ABB RobotStudio station: InjectorSetUp.rsstnx

Station InjectorSetUp (saved by RobotStudio 24.4.11080.0)
Controller IRB4600_60_205_2
  mechanical unit ROB_1: IRB4600_60_205_C_01, 6 joints, base frame (0, 0, 0) mm
Layout (positions relative to the parent item):
  - 1. AttacherBlackL [smart component, from Components\Attacher.rslib] at (-1000, 0, 0) mm
      properties: Parent=MoldGripper; Flange=0; Child=1. BlackL; Mount=false; Offset=[0 0 0]; Orientation=[0 0 0]
  - 1. TakeSensorBlackL [smart component, from Components\LineSensor.rslib] at (-1000, 295, -84.5) mm
      properties: Start=[0.95 1.25 1.44146]; End=[1.05 1.25 1.44146]; Length=0.1; Radius=0; Tag=(none); SensedPart=(none); SensedPoint=[0 0 0]
    - _sensorPart_ [part], size 100 x 0 x 0 mm
  - 1. PosBlackL [smart component, from Components\Positioner.rslib] at (-1000, 300, 0) mm
      properties: Object=1. BlackL; Position=[-0.25 1.55 1.5]; Orientation=[0 0 0]; Reference=Global; ReferenceObject=(none)
  - 1. DetacherBlackL [smart component, from Components\Detacher.rslib] at (-1000, 300, 0) mm
      properties: Child=1. BlackL; KeepPosition=true
  - 0. DropSensorBaseL [smart component, from Components\LineSensor.rslib] at (-1500, -37.49, 0) mm
      properties: Start=[3.2 0.43748 1.53501]; End=[2.7 0.43748 1.53501]; Length=0.5; Radius=0; Tag=(none); SensedPart=(none); SensedPoint=[0 0 0]
    - _sensorPart_ [part], size 500 x 0 x 0 mm
  - 1. PosBlackR [smart component, from Components\Positioner.rslib] at (-1000, -300, 0) mm
      properties: Object=1. BlackR; Position=[0.25 -1.55 1.5]; Orientation=[0 0 3.14159265358979]; Reference=Global; ReferenceObject=(none)
  - 1. AttacherBlackR [smart component, from Components\Attacher.rslib] at (-1000, -100, 0) mm
      properties: Parent=MoldGripper; Flange=0; Child=1. BlackR; Mount=false; Offset=[0 0 0]; Orientation=[0 0 0]
  - 1. TakeSensorBlackR [smart component, from Components\LineSensor.rslib] at (-1150, -300, -91.46) mm
      properties: Start=[1.1 -1.245 1.44842]; End=[1.2 -1.245 1.44842]; Length=0.1; Radius=0; Tag=(none); SensedPart=(none); SensedPoint=[0 0 0]
    - _sensorPart_ [part], size 100 x 0 x 0 mm
  - 0. TakeSensorBaseR [smart component, from Components\LineSensor.rslib] at (-1500, -800, -91.46) mm
      properties: Start=[3 0.605 1.54842]; End=[2.9 0.605 1.54842]; Length=0.0999999999999996; Radius=0; Tag=(none); SensedPart=(none); SensedPoint=[0 0 0]
    - _sensorPart_ [part], size 100 x 0 x 0 mm
  - 1. DetacherBlackR [smart component, from Components\Detacher.rslib] at (-1000, -300, 0) mm
      properties: Child=1. BlackR; KeepPosition=true
  - 2. AttacherRedL [smart component, from Components\Attacher.rslib] at (-1420, 300, 0) mm
      properties: Parent=MoldGripper; Flange=0; Child=2. RedL; Mount=false; Offset=[0 0 0]; Orientation=[0 0 0]
  - 2. TakeSensorRedL [smart component, from Components\LineSensor.rslib] at (-1150, 300, -91.46) mm
      properties: Start=[1.1 1.245 0.94842]; End=[1.2 1.245 0.94842]; Length=0.1; Radius=0; Tag=(none); SensedPart=(none); SensedPoint=[0 0 0]
    - _sensorPart_ [part], size 100 x 0 x 0 mm
  - 2. PosRedL [smart component, from Components\Positioner.rslib] at (-1420, 100, 0) mm
      properties: Object=2. RedL; Position=[-0.25 1.55 1]; Orientation=[0 0 0]; Reference=Global; ReferenceObject=(none)
  - 2. DetacherRedL [smart component, from Components\Detacher.rslib] at (-1420, 300, 0) mm
      properties: Child=2. RedL; KeepPosition=true
  - 2. PosRedR [smart component, from Components\Positioner.rslib] at (-1420, -300, 0) mm
      properties: Object=2. RedR; Position=[0.25 -1.55 1]; Orientation=[0 0 3.14159265358979]; Reference=Global; ReferenceObject=(none)
  - 2. AttacherRedR [smart component, from Components\Attacher.rslib] at (-1420, -300, 0) mm
      properties: Parent=MoldGripper; Flange=0; Child=2. RedR; Mount=false; Offset=[0 0 0]; Orientation=[0 0 0]
  - 2. TakeSensorRedR [smart component, from Components\LineSensor.rslib] at (-1570, -300, -91.46) mm
      properties: Start=[1.52 -1.245 0.94842]; End=[1.62 -1.245 0.94842]; Length=0.1; Radius=0; Tag=(none); SensedPart=(none); SensedPoint=[0 0 0]
    - _sensorPart_ [part], size 100 x 0 x 0 mm
  - 2. DetacherRedR [smart component, from Components\Detacher.rslib] at (-1420, -300, 0) mm
      properties: Child=2. RedR; KeepPosition=true
  - 3. AttacherBlueL [smart component, from Components\Attacher.rslib] at (-1840, 300, 0) mm
      properties: Parent=MoldGripper; Flange=0; Child=3. BlueL; Mount=false; Offset=[0 0 0]; Orientation=[0 0 0]
  - 3. TakeSensorBlueL [smart component, from Components\LineSensor.rslib] at (-1150, 300, -91.46) mm
      properties: Start=[1.1 1.245 0.44842]; End=[1.2 1.245 0.44842]; Length=0.1; Radius=0; Tag=(none); SensedPart=(none); SensedPoint=[0 0 0]
    - _sensorPart_ [part], size 100 x 0 x 0 mm
  - 3. PosBlueL [smart component, from Components\Positioner.rslib] at (-1840, 300, 0) mm
      properties: Object=3. BlueL; Position=[-0.25 1.55 0.5]; Orientation=[0 0 0]; Reference=Global; ReferenceObject=(none)
  - 3. DetacherBlueL [smart component, from Components\Detacher.rslib] at (-1840, 300, 0) mm
      properties: Child=3. BlueL; KeepPosition=true
  - 3. PosBlueR [smart component, from Components\Positioner.rslib] at (-1840, -300, 0) mm
      properties: Object=3. BlueR; Position=[0.25 -1.55 0.5]; Orientation=[0 0 3.14159265358979]; Reference=Global; ReferenceObject=(none)
  - 3. AttacherBlueR [smart component, from Components\Attacher.rslib] at (-1840, -300, 0) mm
      properties: Parent=MoldGripper; Flange=0; Child=3. BlueR; Mount=false; Offset=[0 0 0]; Orientation=[0 0 0]
  - 3. TakeSensorBlueR [smart component, from Components\LineSensor.rslib] at (-1990, -300, -91.46) mm
      properties: Start=[1.94 -1.245 0.44842]; End=[2.04 -1.245 0.44842]; Length=0.1; Radius=0; Tag=(none); SensedPart=(none); SensedPoint=[0 0 0]
    - _sensorPart_ [part], size 100 x 0 x 0 mm
  - 3. DetacherBlueR [smart component, from Components\Detacher.rslib] at (-1840, -300, 0) mm
      properties: Child=3. BlueR; KeepPosition=true
  - InjectionMachine [part] at (900, 1700, 0) mm, size 1314.8 x 3413.3 x 1819.5 mm
  - ClosePressFunction [smart component, from Components\JointMover.rslib] at (-1000, 0, 0) mm
      properties: Mechanism=Press; Relative=false; Duration=0.5; J1=0.4
  - OpenPressFunction [smart component, from Components\JointMover.rslib] at (-1000, 0, 0) mm
      properties: Mechanism=Press; Relative=false; Duration=0.5; J1=0
  - 0. DropSensorBaseR [smart component, from Components\LineSensor.rslib] at (-1500, -800, 50) mm
      properties: Start=[3.2 0.40001 1.48501]; End=[2.7 0.40001 1.48501]; Length=0.5; Radius=0; Tag=(none); SensedPart=2. RedR; SensedPoint=[1.20000036621094 -0.399989990234375 1.53501000976562]
    - _sensorPart_ [part], size 500 x 0 x 0 mm
  - 0. AttacherBaseRBlackR [smart component, from Components\Attacher.rslib] at (-1300, 0, 0) mm
      properties: Parent=Press; Flange=0; Child=1. BlackR; Mount=false; Offset=[0 0 0]; Orientation=[0 0 0]
  - 0. AttacherBaseRBlueR [smart component, from Components\Attacher.rslib] at (-1300, 0, 0) mm
      properties: Parent=Press; Flange=0; Child=3. BlueR; Mount=false; Offset=[0 0 0]; Orientation=[0 0 0]
  - 0. AttacherBaseRedR [smart component, from Components\Attacher.rslib] at (-1300, 0, 0) mm
      properties: Parent=Press; Flange=0; Child=2. RedR; Mount=false; Offset=[0 0 0]; Orientation=[0 0 0]
  - BlackRight [smart component, from Components\LogicGate.rslib]
      properties: Operator=AND; Delay=0
  - RedRight [smart component, from Components\LogicGate.rslib]
      properties: Operator=AND; Delay=0
  - BlueRight [smart component, from Components\LogicGate.rslib]
      properties: Operator=AND; Delay=0
  - 1. VolumeBlackR [smart component, from Components\VolumeSensor.rslib] at (-1020, -280, -20) mm
      properties: CornerPoint=[0.75 -1.25 1.1]; Orientation=[0 0 -1.5707963267949]; Length=0.24; Width=0.54; Height=0.44; Tag=(none); PartialHit=false; SensedPart=1. BlackR
    - _sensorPart_ [part], size 540 x 240 x 440 mm
  - BlackRight [smart component, from Components\LogicGate.rslib]
      properties: Operator=NOT; Delay=0
  - 2. VolumeRedR [smart component, from Components\VolumeSensor.rslib] at (-1020, -280, -520) mm
      properties: CornerPoint=[0.75 -1.25 1.1]; Orientation=[0 0 -1.5707963267949]; Length=0.24; Width=0.54; Height=0.44; Tag=(none); PartialHit=false; SensedPart=(none)
    - _sensorPart_ [part], size 540 x 240 x 440 mm
  - 3. VolumeBlueR [smart component, from Components\VolumeSensor.rslib] at (-1020, -280, -1020) mm
      properties: CornerPoint=[0.75 -1.25 1.1]; Orientation=[0 0 -1.5707963267949]; Length=0.24; Width=0.54; Height=0.44; Tag=(none); PartialHit=false; SensedPart=3. BlueR
    - _sensorPart_ [part], size 540 x 240 x 440 mm
  - RedRight [smart component, from Components\LogicGate.rslib]
      properties: Operator=NOT; Delay=0
  - BlueRight [smart component, from Components\LogicGate.rslib]
      properties: Operator=NOT; Delay=0
  - 0. VolumeBaseR [smart component, from Components\VolumeSensor.rslib] at (-1800, 840, 0) mm
      properties: CornerPoint=[2.99 -1.03 1.19]; Orientation=[0 0 -1.5707963267949]; Length=0.215; Width=0.515; Height=0.415; Tag=(none); PartialHit=false; SensedPart=2. RedR
    - _sensorPart_ [part], size 515 x 215 x 415 mm
  - 0. VolumeBaseL [smart component, from Components\VolumeSensor.rslib] at (-1800, 1000, 0) mm
      properties: CornerPoint=[3.51 -0.81 1.19]; Orientation=[0 0 1.5707963267949]; Length=0.215; Width=0.515; Height=0.415; Tag=(none); PartialHit=false; SensedPart=(none)
    - _sensorPart_ [part], size 515 x 215 x 415 mm
  - TakeRight [smart component, from Components\LogicGate.rslib]
      properties: Operator=AND; Delay=0
  - TakeRight [smart component, from Components\LogicGate.rslib]
      properties: Operator=NOT; Delay=0
  - BaseBlackRight [smart component, from Components\LogicGate.rslib]
      properties: Operator=AND; Delay=0
  - 0. PosBaseBlackR [smart component, from Components\Positioner.rslib] at (-1300, 0, 0) mm
      properties: Object=1. BlackR; Position=[1.7 -0.2 1.6]; Orientation=[0 0 -3.14159265358979]; Reference=Global; ReferenceObject=(none)
  - 0. PosBaseBlackL [smart component, from Components\Positioner.rslib] at (-1300, 0, 0) mm
      properties: Object=1. BlackL; Position=[1.2 0.2 1.6]; Orientation=[0 0 0]; Reference=Global; ReferenceObject=(none)
  - TakeLeft [smart component, from Components\LogicGate.rslib]
      properties: Operator=AND; Delay=0
  - BaseBlackLeft [smart component, from Components\LogicGate.rslib]
      properties: Operator=AND; Delay=0
  - 0. TakeSensorBaseL [smart component, from Components\LineSensor.rslib] at (-1500, -420, -91.46) mm
      properties: Start=[3 0.615 1.54842]; End=[2.9 0.615 1.54842]; Length=0.1; Radius=0; Tag=(none); SensedPart=(none); SensedPoint=[0 0 0]
    - _sensorPart_ [part], size 100 x 0 x 0 mm
  - 1. VolumeBlackL [smart component, from Components\VolumeSensor.rslib] at (-880, 280, -20) mm
      properties: CornerPoint=[1.15 1.25 1.1]; Orientation=[0 0 1.5707963267949]; Length=0.24; Width=0.54; Height=0.44; Tag=(none); PartialHit=false; SensedPart=1. BlackL
    - _sensorPart_ [part], size 540 x 240 x 440 mm
  - 2. VolumeRedL [smart component, from Components\VolumeSensor.rslib] at (-880, 280, -520) mm
      properties: CornerPoint=[1.15 1.25 1.1]; Orientation=[0 0 1.5707963267949]; Length=0.24; Width=0.54; Height=0.44; Tag=(none); PartialHit=false; SensedPart=(none)
    - _sensorPart_ [part], size 540 x 240 x 440 mm
  - 3. VolumeBlueL [smart component, from Components\VolumeSensor.rslib] at (-880, 280, -1020) mm
      properties: CornerPoint=[1.15 1.25 1.1]; Orientation=[0 0 1.5707963267949]; Length=0.24; Width=0.54; Height=0.44; Tag=(none); PartialHit=false; SensedPart=3. BlueL
    - _sensorPart_ [part], size 540 x 240 x 440 mm
  - BlackLeft [smart component, from Components\LogicGate.rslib]
      properties: Operator=NOT; Delay=0
  - RedLeft [smart component, from Components\LogicGate.rslib]
      properties: Operator=NOT; Delay=0
  - BlueLeft [smart component, from Components\LogicGate.rslib]
      properties: Operator=NOT; Delay=0
  - 1. DropSensorBlackL [smart component, from Components\LineSensor.rslib] at (-1000, -221.01, 0) mm
      properties: Start=[0.75 1.971 1.436]; End=[0.85 1.971 1.436]; Length=0.1; Radius=0; Tag=(none); SensedPart=1. BlackL; SensedPoint=[-0.249999877929688 1.74998999023437 1.436]
    - _sensorPart_ [part], size 100 x 0 x 0 mm
  - 1. DropSensorBlackR [smart component, from Components\LineSensor.rslib] at (-1200, -820.98, 0) mm, rotated rx 0 ry 0.01 rz 0 deg
      properties: Start=[1.44974952316885 -0.92901 1.43525305088395]; End=[0.949749530784283 -0.92901 1.4351657844218]; Length=0.5; Radius=0; Tag=(none); SensedPart=1. BlackR; SensedPoint=[0.25 -1.74998999023437 1.435]
    - _sensorPart_ [part], size 500 x 0 x 0.1 mm
  - 2. DropSensorRedR [smart component, from Components\LineSensor.rslib] at (-1200, -820.98, -500) mm, rotated rx 0 ry 0.01 rz 0 deg
      properties: Start=[1.44974952316885 -0.92901 1.43525305088395]; End=[0.949749530784283 -0.92901 1.4351657844218]; Length=0.5; Radius=0; Tag=(none); SensedPart=(none); SensedPoint=[0 0 0]
    - _sensorPart_ [part], size 500 x 0 x 0.1 mm
  - 2. DropSensorRedL [smart component, from Components\LineSensor.rslib] at (-1000, -221.01, -500) mm
      properties: Start=[0.75 1.971 1.435]; End=[1.25 1.971 1.435]; Length=0.5; Radius=0; Tag=(none); SensedPart=(none); SensedPoint=[0 0 0]
    - _sensorPart_ [part], size 500 x 0 x 0 mm
  - 3. DropSensorBlueR [smart component, from Components\LineSensor.rslib] at (-1200, -820.98, -1000) mm, rotated rx 0 ry 0.01 rz 0 deg
      properties: Start=[1.44974952316885 -0.92901 1.43525305088395]; End=[0.949749530784283 -0.92901 1.4351657844218]; Length=0.5; Radius=0; Tag=(none); SensedPart=3. BlueR; SensedPoint=[0.25 -1.74998999023437 0.435]
    - _sensorPart_ [part], size 500 x 0 x 0.1 mm
  - 3. DropSensorBlueL [smart component, from Components\LineSensor.rslib] at (-1000, -221.01, -1000) mm
      properties: Start=[0.75 1.971 1.435]; End=[1.25 1.971 1.435]; Length=0.5; Radius=0; Tag=(none); SensedPart=3. BlueL; SensedPoint=[0.249999969482422 1.74998999023437 0.435]
    - _sensorPart_ [part], size 500 x 0 x 0 mm
  - CloseSecurityTimer [smart component, from Components\Timer.rslib] at (-1000, 0, 0) mm
      properties: StartTime=1; Interval=0; Repeat=false; CurrentTime=0
  - InjectionCycleTimer [smart component, from Components\Timer.rslib]
      properties: StartTime=15.5; Interval=0; Repeat=false; CurrentTime=0
  - LogicSRLatch [smart component, from Components\LogicSRLatch.rslib]
  - BaseRedRight [smart component, from Components\LogicGate.rslib]
      properties: Operator=AND; Delay=0
  - BaseRedLeft [smart component, from Components\LogicGate.rslib]
      properties: Operator=AND; Delay=0
  - BaseBlueRight [smart component, from Components\LogicGate.rslib]
      properties: Operator=AND; Delay=0
  - BaseBlueLeft [smart component, from Components\LogicGate.rslib]
      properties: Operator=AND; Delay=0
  - ResetTimerAux [smart component, from Components\Timer.rslib] at (-600, 0, 0) mm
      properties: StartTime=0.1; Interval=0; Repeat=false; CurrentTime=192.816
  - IRB4600_60_205_C_01 [mechanism, from %ABB.RobotStudio.Models.IRB4600%\IRB4600_60_205_C_G_01.rslib] at (0, 0, 0) mm; joint values [1.5708, 0.4406, 0.2713, 0, -0.7118, 0] (rad or m)
  - OutMold1 [part] at (1510.58, -210, 320) mm, size 400 x 400 x 50 mm
  - FirstConveyor [part] at (1000, 190, 200) mm, size 2000 x 500 x 900 mm
  - MovementOutMold1 [smart component, from Components\MoveAlongCurve.rslib]
      properties: Object=OutMold1; WirePart=WayOutMold1; Speed=0.5; KeepOrientation=false; StartDistance=0; ResetPosition=true; StartPosition=[[1 0 0 0] [0 1 0 0] [0 0 1 0] [1.74 -0.21 0.32 1]]
  - MovementOutMold2 [smart component, from Components\MoveAlongCurve.rslib]
      properties: Object=OutMold2; WirePart=WayOutMold2; Speed=0.5; KeepOrientation=false; StartDistance=0; ResetPosition=false; StartPosition=[[1 0 0 0] [0 1 0 0] [0 0 1 0] [0 0 0 1]]
  - WayOutMold1 [part] at (-800, 0, 0) mm, size 240.6 x 0 x 0 mm
  - HideOutMold1 [smart component, from Components\Hide.rslib]
      properties: Object=OutMold1
  - HideOutMold2 [smart component, from Components\Hide.rslib]
      properties: Object=OutMold2
  - OutMold2 [part] at (2300.58, -211, 545) mm, rotated rx 0 ry -30 rz 0 deg, size 400 x 400 x 50 mm
  - ShowOutMold1 [smart component, from Components\Show.rslib] at (-600, 0, 0) mm
      properties: Object=OutMold1
  - ShowOutMold2 [smart component, from Components\Show.rslib] at (-600, 0, 0) mm
      properties: Object=OutMold2
  - WayOutMold2 [part] at (-600, 0, 0) mm, size 958.1 x 0 x 555.7 mm
  - PositionerOutMold1 [smart component, from Components\Positioner.rslib] at (-600, 0, 0) mm
      properties: Object=OutMold1; Position=[1.510578 -0.21 0.32]; Orientation=[0 0 0]; Reference=Global; ReferenceObject=(none)
  - PositionerOutMold2 [smart component, from Components\Positioner.rslib] at (-600, 0, 0) mm
      properties: Object=OutMold2; Position=[2.300578 -0.211 0.545]; Orientation=[0 -0.523598775598299 0]; Reference=Global; ReferenceObject=(none)
  - BlueColorOutMold1 [smart component, from Components\Highlighter.rslib]
      properties: Object=OutMold1; Color=[0 150 255]; Opacity=255
  - BlueColorOutMold2 [smart component, from Components\Highlighter.rslib]
      properties: Object=OutMold2; Color=[0 150 255]; Opacity=255
  - RedColorOutMold1 [smart component, from Components\Highlighter.rslib] at (-600, 0, 0) mm
      properties: Object=OutMold1; Color=[255 0 0]; Opacity=255
  - RedColorOutMold2 [smart component, from Components\Highlighter.rslib] at (-600, 0, 0) mm
      properties: Object=OutMold2; Color=[255 0 0]; Opacity=255
  - RedColorCount [smart component, from Components\Comparer.rslib] at (-600, 0, 0) mm
      properties: ValueA=2; Operator===; ValueB=1
  - CoreColorCounter [smart component, from Components\Counter.rslib]
      properties: Count=2
  - BlueColorCount [smart component, from Components\Comparer.rslib]
      properties: ValueA=2; Operator===; ValueB=2
  - ResetCoreCounter [smart component, from Components\Comparer.rslib] at (-600, 0, 0) mm
      properties: ValueA=2; Operator===; ValueB=3
  - OutMold1Sensor [smart component, from Components\LineSensor.rslib] at (-600, 0, 0) mm
      properties: Start=[1.910578 0.19 0.38]; End=[1.910578 -0.21 0.38]; Length=0.4; Radius=0; Tag=(none); SensedPart=(none); SensedPoint=[0 0 0]
    - _sensorPart_ [part], size 0 x 400 x 0 mm
  - RealOut [part] at (1610.58, -40, 1550) mm, rotated rx -90 ry 0 rz 0 deg, size 400 x 400 x 50 mm
  - MovementRealOutMold [smart component, from Components\LinearMover2.rslib]
      properties: Object=RealOut; Direction=[0 0 -0.001]; Distance=0.8; Duration=0.404; Reference=Global; ReferenceObject=(none)
  - PositionerRealOut [smart component, from Components\Positioner.rslib] at (-600, 0, 0) mm
      properties: Object=RealOut; Position=[1.610578 -0.04 1.55]; Orientation=[-1.5707963267949 0 0]; Reference=Global; ReferenceObject=(none)
  - ShowRealOutMold [smart component, from Components\Show.rslib] at (-600, 0, 0) mm
      properties: Object=RealOut
  - HideRealOut [smart component, from Components\Hide.rslib]
      properties: Object=RealOut
  - OpenPressAuxFunction [smart component, from Components\JointMover.rslib] at (-1000, 0, 0) mm
      properties: Mechanism=Press; Relative=false; Duration=0.5; J1=0
  - RedColorRealMold [smart component, from Components\Highlighter.rslib] at (-600, 0, 0) mm
      properties: Object=RealOut; Color=[255 0 0]; Opacity=255
  - BlueColorRealMold [smart component, from Components\Highlighter.rslib] at (-600, 0, 0) mm
      properties: Object=RealOut; Color=[0 150 255]; Opacity=255
  - IRC5_Single-Cabinet [part, from %ABB.RobotStudio.Models.IRC5%\IRC5_Single-Cabinet.rslib] at (-3450, 450, 100) mm, rotated rx 90 ry 0 rz -90 deg
  - FlexPendant [part, from %ABB.RobotStudio.Models.IRC5%\FlexPendant.rslib] at (-3350, 630, 990) mm, rotated rx -27.17 ry 5.43 rz -119.59 deg
  - EnablingSwitch [part] at (-3520, 650, 920) mm, rotated rx 0 ry 0 rz 180 deg, size 62.9 x 279 x 47.8 mm
  - MoldGripper [mechanism] at (0, 1535, 814.49) mm, rotated rx 0 ry 90 rz 90 deg
      TCP MoldGripper at (0, -85, -10.5) mm, rotated rx 0 ry -90 rz 90 deg
      links: EndEffector
  - 0. BaseMoldL [part] at (-300, 0, 4000) mm, size 500 x 200 x 400 mm
  - Press [mechanism] at (-300, 0, 0) mm; joint values [0] (rad or m)
      links: Link1, Link2
  - 3. BlueL [part] at (-250, 1550, 498.43) mm, size 500 x 200 x 400 mm
  - 2. RedL [part] at (-250, 1550, 1019.95) mm, size 500 x 200 x 400 mm
  - 1. BlackL [part] at (-250, 1550, 1500.71) mm, size 500 x 200 x 400 mm
  - 1. BlackR [part] at (250, -1550, 1500) mm, rotated rx 0 ry 0 rz 180 deg, size 500 x 200 x 400 mm
  - 2. RedR [part] at (1700, -200, 1599.37) mm, rotated rx 0 ry 0 rz -180 deg, size 500 x 200 x 400 mm
  - 3. BlueR [part] at (250, -1550, 500) mm, rotated rx 0 ry 0 rz 180 deg, size 500 x 200 x 400 mm
  - MoldStore [part] at (285, 1550, 0) mm, rotated rx 0 ry 0 rz 90 deg, size 300 x 610 x 1600 mm
  - MoldStore_2 [part] at (-285, -1550, 0) mm, rotated rx 0 ry 0 rz -90 deg, size 300 x 610 x 1600 mm
  - Fence_3 [graphiccomponentgroup]
    - Segment 1 [part], size 169.7 x 169.7 x 1400 mm
    - Segment 2 [part], size 316.7 x 1054.9 x 1400 mm
    - Segment 3 [part], size 169.7 x 1684.9 x 1400 mm
    - Segment 3 [part], size 169.7 x 1684.9 x 1400 mm
    - Segment 3 [part], size 169.7 x 1684.9 x 1400 mm
  - Fence_2 [graphiccomponentgroup]
    - Segment 1 [part], size 169.7 x 169.7 x 1400 mm
    - Segment 2 [part], size 1959.9 x 169.7 x 1400 mm
    - Segment 2 [part], size 1959.9 x 169.7 x 1400 mm
  - Fence [graphiccomponentgroup]
    - Segment 1 [part], size 169.7 x 169.7 x 1400 mm
    - Segment 2 [part], size 1959.9 x 169.7 x 1400 mm
    - Segment 2 [part], size 1959.9 x 169.7 x 1400 mm
  - Fence_6 [graphiccomponentgroup]
    - Segment 1 [part], size 169.7 x 169.7 x 2000 mm
    - Segment 2 [part], size 169.7 x 1134.9 x 2000 mm
    - Segment 2 [part], size 169.7 x 1134.9 x 2000 mm
  - Fence_4 [graphiccomponentgroup]
    - Segment 1 [part], size 169.7 x 169.7 x 2000 mm
    - Segment 2 [part], size 169.7 x 1134.9 x 2000 mm
    - Segment 2 [part], size 169.7 x 1134.9 x 2000 mm
  - Fence_5 [graphiccomponentgroup]
    - Segment 1 [part], size 169.7 x 169.7 x 1400 mm
    - Segment 2 [part], size 169.7 x 169.7 x 1400 mm
  - Pieza_3 [part], size 15 x 940 x 15 mm
  - Pieza_4 [part] at (0, 0, 500) mm, size 15 x 940 x 15 mm
  - Pieza_5 [part] at (0, 0, -500) mm, size 15 x 940 x 15 mm
  - ControlPanel [part] at (-3165, 1650, 600) mm, rotated rx 0 ry 0 rz -90 deg, size 600 x 300 x 800 mm
  - ModeSelecting1 [smart component, from Components\LogicMux.rslib]
  - ModeSelecting2 [smart component, from Components\LogicMux.rslib]
  - ModeCounter [smart component, from Components\Counter.rslib]
      properties: Count=5
Attachment: MoldGripper is attached to IRB4600_60_205_C_01 / Link6
Attachment: 2. RedR is attached to Press / Link2
Attachment: 2. RedL is attached to MoldGripper / EndEffector
Station signals: DI Digital1, DI Digital2
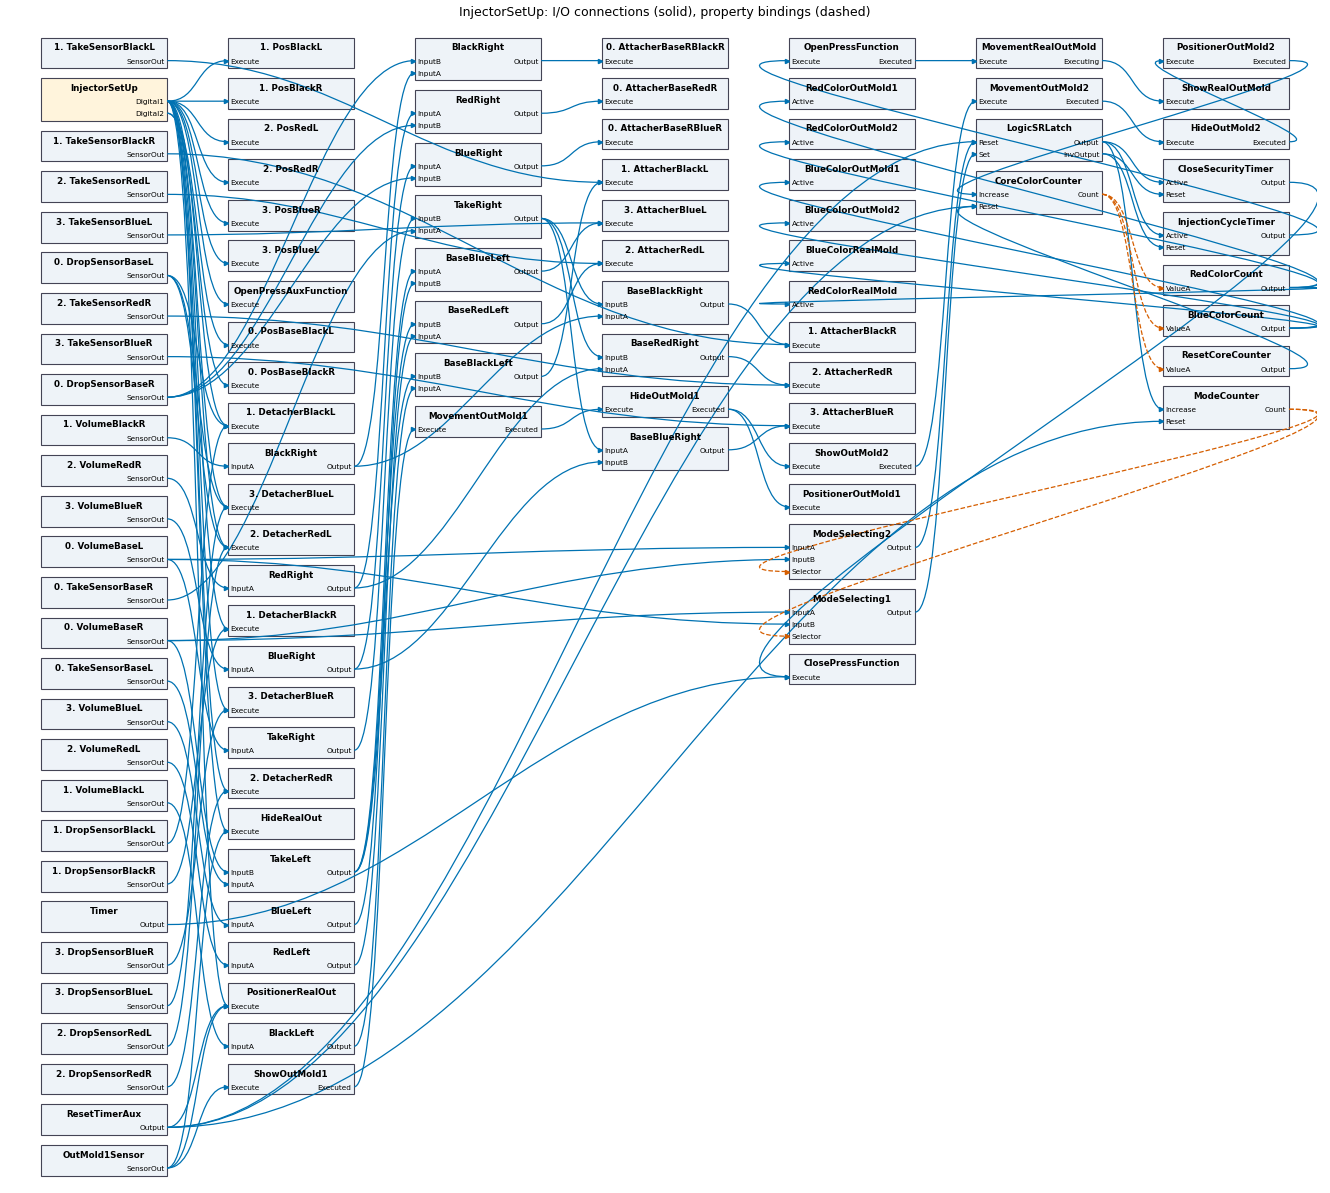
Station logic (signal -> signal, property => property):
  1. TakeSensorBlackL.SensorOut -> 1. AttacherBlackL.Execute
  InjectorSetUp.Digital1 -> 1. PosBlackL.Execute
  InjectorSetUp.Digital1 -> 1. DetacherBlackL.Execute
  InjectorSetUp.Digital1 -> 1. PosBlackR.Execute
  1. TakeSensorBlackR.SensorOut -> 1. AttacherBlackR.Execute
  InjectorSetUp.Digital1 -> 1. DetacherBlackR.Execute
  InjectorSetUp.Digital1 -> 2. DetacherRedL.Execute
  InjectorSetUp.Digital1 -> 3. DetacherBlueL.Execute
  InjectorSetUp.Digital1 -> 2. DetacherRedR.Execute
  InjectorSetUp.Digital1 -> 3. DetacherBlueR.Execute
  2. TakeSensorRedL.SensorOut -> 2. AttacherRedL.Execute
  3. TakeSensorBlueL.SensorOut -> 3. AttacherBlueL.Execute
  0. DropSensorBaseL.SensorOut -> 1. DetacherBlackL.Execute
  0. DropSensorBaseL.SensorOut -> 2. DetacherRedL.Execute
  0. DropSensorBaseL.SensorOut -> 3. DetacherBlueL.Execute
  2. TakeSensorRedR.SensorOut -> 2. AttacherRedR.Execute
  3. TakeSensorBlueR.SensorOut -> 3. AttacherBlueR.Execute
  InjectorSetUp.Digital1 -> 2. PosRedL.Execute
  InjectorSetUp.Digital1 -> 2. PosRedR.Execute
  InjectorSetUp.Digital1 -> 3. PosBlueR.Execute
  InjectorSetUp.Digital1 -> 3. PosBlueL.Execute
  0. DropSensorBaseR.SensorOut -> BlackRight.InputB
  1. VolumeBlackR.SensorOut -> BlackRight.InputA
  BlackRight.Output -> BlackRight.InputA
  BlackRight.Output -> 0. AttacherBaseRBlackR.Execute
  2. VolumeRedR.SensorOut -> RedRight.InputA
  RedRight.Output -> RedRight.InputA
  RedRight.Output -> 0. AttacherBaseRedR.Execute
  3. VolumeBlueR.SensorOut -> BlueRight.InputA
  BlueRight.Output -> BlueRight.InputA
  0. DropSensorBaseR.SensorOut -> BlueRight.InputB
  0. DropSensorBaseR.SensorOut -> RedRight.InputB
  BlueRight.Output -> 0. AttacherBaseRBlueR.Execute
  0. VolumeBaseL.SensorOut -> TakeRight.InputA
  TakeRight.Output -> TakeRight.InputB
  0. TakeSensorBaseR.SensorOut -> TakeRight.InputA
  TakeRight.Output -> BaseBlackRight.InputB
  BaseBlackRight.Output -> 1. AttacherBlackR.Execute
  InjectorSetUp.Digital2 -> 0. PosBaseBlackL.Execute
  InjectorSetUp.Digital2 -> 0. PosBaseBlackR.Execute
  0. VolumeBaseR.SensorOut -> TakeLeft.InputB
  0. TakeSensorBaseL.SensorOut -> TakeLeft.InputA
  TakeLeft.Output -> BaseBlackLeft.InputB
  3. VolumeBlueL.SensorOut -> BlueLeft.InputA
  2. VolumeRedL.SensorOut -> RedLeft.InputA
  1. VolumeBlackL.SensorOut -> BlackLeft.InputA
  BlackLeft.Output -> BaseBlackLeft.InputA
  BaseBlackLeft.Output -> 1. AttacherBlackL.Execute
  BlackRight.Output -> BaseBlackRight.InputA
  1. DropSensorBlackL.SensorOut -> 1. DetacherBlackL.Execute
  1. DropSensorBlackR.SensorOut -> 1. DetacherBlackR.Execute
  Timer.Output -> ClosePressFunction.Execute
  CloseSecurityTimer.Output -> ClosePressFunction.Execute
  InjectionCycleTimer.Output -> OpenPressFunction.Execute
  LogicSRLatch.Output -> CloseSecurityTimer.Active
  LogicSRLatch.Output -> InjectionCycleTimer.Active
  LogicSRLatch.InvOutput -> InjectionCycleTimer.Reset
  LogicSRLatch.InvOutput -> CloseSecurityTimer.Reset
  3. DropSensorBlueR.SensorOut -> 3. DetacherBlueR.Execute
  3. DropSensorBlueL.SensorOut -> 3. DetacherBlueL.Execute
  2. DropSensorRedL.SensorOut -> 2. DetacherRedL.Execute
  2. DropSensorRedR.SensorOut -> 2. DetacherRedR.Execute
  TakeLeft.Output -> BaseRedLeft.InputB
  RedLeft.Output -> BaseRedLeft.InputA
  BaseRedLeft.Output -> 2. AttacherRedL.Execute
  TakeRight.Output -> BaseRedRight.InputB
  RedRight.Output -> BaseRedRight.InputA
  BaseRedRight.Output -> 2. AttacherRedR.Execute
  TakeLeft.Output -> BaseBlueLeft.InputA
  BlueLeft.Output -> BaseBlueLeft.InputB
  BaseBlueLeft.Output -> 3. AttacherBlueL.Execute
  TakeRight.Output -> BaseBlueRight.InputA
  BlueRight.Output -> BaseBlueRight.InputB
  BaseBlueRight.Output -> 3. AttacherBlueR.Execute
  ResetTimerAux.Output -> LogicSRLatch.Reset
  HideOutMold1.Executed -> ShowOutMold2.Execute
  ShowOutMold1.Executed -> MovementOutMold1.Execute
  ShowOutMold2.Executed -> MovementOutMold2.Execute
  MovementOutMold1.Executed -> HideOutMold1.Execute
  HideOutMold1.Executed -> PositionerOutMold1.Execute
  HideOutMold2.Executed -> PositionerOutMold2.Execute
  MovementOutMold2.Executed -> HideOutMold2.Execute
  PositionerOutMold2.Executed -> CoreColorCounter.Increase
  RedColorCount.Output -> RedColorOutMold1.Active
  RedColorCount.Output -> RedColorOutMold2.Active
  BlueColorCount.Output -> BlueColorOutMold1.Active
  BlueColorCount.Output -> BlueColorOutMold2.Active
  ResetTimerAux.Output -> CoreColorCounter.Reset
  ResetCoreCounter.Output -> CoreColorCounter.Reset
  OutMold1Sensor.SensorOut -> PositionerRealOut.Execute
  OutMold1Sensor.SensorOut -> ShowOutMold1.Execute
  ResetTimerAux.Output -> PositionerRealOut.Execute
  OpenPressFunction.Executed -> MovementRealOutMold.Execute
  InjectorSetUp.Digital1 -> PositionerRealOut.Execute
  OutMold1Sensor.SensorOut -> HideRealOut.Execute
  MovementRealOutMold.Executing -> ShowRealOutMold.Execute
  InjectorSetUp.Digital1 -> HideRealOut.Execute
  InjectorSetUp.Digital1 -> OpenPressAuxFunction.Execute
  BlueColorCount.Output -> BlueColorRealMold.Active
  RedColorCount.Output -> RedColorRealMold.Active
  0. VolumeBaseL.SensorOut -> ModeSelecting2.InputA
  ModeSelecting2.Output -> LogicSRLatch.Reset
  0. VolumeBaseR.SensorOut -> ModeSelecting2.InputB
  0. VolumeBaseR.SensorOut -> ModeSelecting1.InputA
  ModeSelecting1.Output -> LogicSRLatch.Set
  0. VolumeBaseL.SensorOut -> ModeSelecting1.InputB
  LogicSRLatch.Output -> ModeCounter.Increase
  ResetTimerAux.Output -> ModeCounter.Reset
  CoreColorCounter.Count => RedColorCount.ValueA
  CoreColorCounter.Count => BlueColorCount.ValueA
  CoreColorCounter.Count => ResetCoreCounter.ValueA
  ModeCounter.Count => ModeSelecting2.Selector
  ModeCounter.Count => ModeSelecting1.Selector
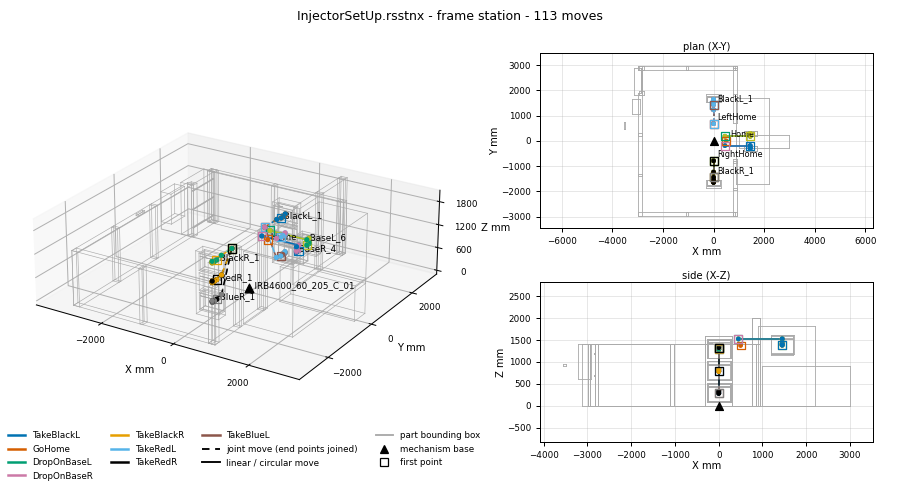
[picture p0: tool path of InjectorSetUp.rsstnx in frame station, 113 of 114 moves have a stored position in this frame; points joined in program order, loops and branches not executed]
Targets, tools, work objects and paths stored in the station, written as RAPID:
! task T_ROB1
MODULE Module1
  CONST jointtarget Rest:=[[0,-60,60,0,30,0],[9E+09,9E+09,9E+09,9E+09,9E+09,9E+09]];
  PROC GoRest()
    MoveAbsJ Rest,robotSpeed,z100,tool0\WObj:=wobj0;
  ENDPROC
  PROC TakeBlackL()
    MoveJ BlackL_1,robotSpeed,z100,MoldGripper\WObj:=LeftMoldStore;
    MoveL BlackL_2,robotSpeed,fine,MoldGripper\WObj:=LeftMoldStore;
    MoveL BlackL_3,robotSpeed,fine,MoldGripper\WObj:=LeftMoldStore;
    MoveL BlackL_4,robotSpeed,fine,MoldGripper\WObj:=LeftMoldStore;
    MoveL BlackL_5,robotSpeed,fine,MoldGripper\WObj:=LeftMoldStore;
    MoveL BlackL_6,robotSpeed,fine,MoldGripper\WObj:=LeftMoldStore;
    MoveJ LeftHome,robotSpeed,z100,MoldGripper\WObj:=LeftMoldStore;
  ENDPROC
  PROC GoHome()
    MoveJ Home,robotSpeed,z100,MoldGripper\WObj:=BaseMolds;
  ENDPROC
  PROC DropOnBaseL()
    MoveJ BaseL_7,robotSpeed,fine,MoldGripper\WObj:=BaseMolds;
    MoveL BaseL_6,robotSpeed,fine,MoldGripper\WObj:=BaseMolds;
    MoveL BaseL_5,robotSpeed,fine,MoldGripper\WObj:=BaseMolds;
    MoveL BaseL_4,robotSpeed,fine,MoldGripper\WObj:=BaseMolds;
    MoveL BaseL_3,robotSpeed,fine,MoldGripper\WObj:=BaseMolds;
    MoveL BaseL_2,robotSpeed,fine,MoldGripper\WObj:=BaseMolds;
    MoveL BaseL_1,robotSpeed,fine,MoldGripper\WObj:=BaseMolds;
  ENDPROC
  PROC DropOnBaseR()
    MoveJ BaseR_7,robotSpeed,fine,MoldGripper\WObj:=BaseMolds;
    MoveL BaseR_6,robotSpeed,fine,MoldGripper\WObj:=BaseMolds;
    MoveL BaseR_5,robotSpeed,fine,MoldGripper\WObj:=BaseMolds;
    MoveL BaseR_4,robotSpeed,fine,MoldGripper\WObj:=BaseMolds;
    MoveL BaseR_3,robotSpeed,fine,MoldGripper\WObj:=BaseMolds;
    MoveL BaseR_2,robotSpeed,fine,MoldGripper\WObj:=BaseMolds;
    MoveL BaseR_1,robotSpeed,fine,MoldGripper\WObj:=BaseMolds;
  ENDPROC
  PROC TakeBlackR()
    MoveJ BlackR_1,robotSpeed,z100,MoldGripper\WObj:=RightMoldStore;
    MoveL BlackR_2,robotSpeed,fine,MoldGripper\WObj:=RightMoldStore;
    MoveL BlackR_3,robotSpeed,fine,MoldGripper\WObj:=RightMoldStore;
    MoveL BlackR_4,robotSpeed,fine,MoldGripper\WObj:=RightMoldStore;
    MoveL BlackR_5,robotSpeed,fine,MoldGripper\WObj:=RightMoldStore;
    MoveL BlackR_6,robotSpeed,fine,MoldGripper\WObj:=RightMoldStore;
    MoveJ RightHome,robotSpeed,z100,MoldGripper\WObj:=RightMoldStore;
  ENDPROC
  PROC TakeRedL()
    MoveJ RedL_1,robotSpeed,z100,MoldGripper\WObj:=LeftMoldStore;
    MoveL RedL_2,robotSpeed,fine,MoldGripper\WObj:=LeftMoldStore;
    MoveL RedL_3,robotSpeed,fine,MoldGripper\WObj:=LeftMoldStore;
    MoveL RedL_4,robotSpeed,fine,MoldGripper\WObj:=LeftMoldStore;
    MoveL RedL_5,robotSpeed,fine,MoldGripper\WObj:=LeftMoldStore;
    MoveL RedL_6,robotSpeed,fine,MoldGripper\WObj:=LeftMoldStore;
    MoveJ LeftHome,robotSpeed,z100,MoldGripper\WObj:=LeftMoldStore;
  ENDPROC
  PROC TakeRedR()
    MoveJ RedR_1,robotSpeed,z100,MoldGripper\WObj:=RightMoldStore;
    MoveL RedR_2,robotSpeed,fine,MoldGripper\WObj:=RightMoldStore;
    MoveL RedR_3,robotSpeed,fine,MoldGripper\WObj:=RightMoldStore;
    MoveL RedR_4,robotSpeed,fine,MoldGripper\WObj:=RightMoldStore;
    MoveL RedR_5,robotSpeed,fine,MoldGripper\WObj:=RightMoldStore;
    MoveL RedR_6,robotSpeed,fine,MoldGripper\WObj:=RightMoldStore;
    MoveJ RightHome,robotSpeed,z100,MoldGripper\WObj:=RightMoldStore;
  ENDPROC
  PROC TakeBlueL()
    MoveJ BlueL_1,robotSpeed,z100,MoldGripper\WObj:=LeftMoldStore;
    MoveL BlueL_2,robotSpeed,fine,MoldGripper\WObj:=LeftMoldStore;
    MoveL BlueL_3,robotSpeed,fine,MoldGripper\WObj:=LeftMoldStore;
    MoveL BlueL_4,robotSpeed,fine,MoldGripper\WObj:=LeftMoldStore;
    MoveL BlueL_5,robotSpeed,fine,MoldGripper\WObj:=LeftMoldStore;
    MoveL BlueL_6,robotSpeed,fine,MoldGripper\WObj:=LeftMoldStore;
    MoveJ LeftHome,robotSpeed,z100,MoldGripper\WObj:=LeftMoldStore;
  ENDPROC
  PROC TakeBlueR()
    MoveJ BlueR_1,robotSpeed,z100,MoldGripper\WObj:=RightMoldStore;
    MoveL BlueR_2,robotSpeed,fine,MoldGripper\WObj:=RightMoldStore;
    MoveL BlueR_3,robotSpeed,fine,MoldGripper\WObj:=RightMoldStore;
    MoveL BlueR_4,robotSpeed,fine,MoldGripper\WObj:=RightMoldStore;
    MoveL BlueR_5,robotSpeed,fine,MoldGripper\WObj:=RightMoldStore;
    MoveL BlueR_6,robotSpeed,fine,MoldGripper\WObj:=RightMoldStore;
    MoveJ RightHome,robotSpeed,z100,MoldGripper\WObj:=RightMoldStore;
  ENDPROC
  PROC TakeFromBaseL()
    MoveJ BaseL_1,robotSpeed,z100,MoldGripper\WObj:=BaseMolds;
    MoveL BaseL_2,robotSpeed,fine,MoldGripper\WObj:=BaseMolds;
    MoveL BaseL_3,robotSpeed,fine,MoldGripper\WObj:=BaseMolds;
    MoveL BaseL_4,robotSpeed,fine,MoldGripper\WObj:=BaseMolds;
    MoveL BaseL_5,robotSpeed,fine,MoldGripper\WObj:=BaseMolds;
    MoveL BaseL_6,robotSpeed,fine,MoldGripper\WObj:=BaseMolds;
    MoveL BaseL_7,robotSpeed,fine,MoldGripper\WObj:=BaseMolds;
  ENDPROC
  PROC TakeFromBaseR()
    MoveJ BaseR_1,robotSpeed,z100,MoldGripper\WObj:=BaseMolds;
    MoveL BaseR_2,robotSpeed,fine,MoldGripper\WObj:=BaseMolds;
    MoveL BaseR_3,robotSpeed,fine,MoldGripper\WObj:=BaseMolds;
    MoveL BaseR_4,robotSpeed,fine,MoldGripper\WObj:=BaseMolds;
    MoveL BaseR_5,robotSpeed,fine,MoldGripper\WObj:=BaseMolds;
    MoveL BaseR_6,robotSpeed,fine,MoldGripper\WObj:=BaseMolds;
    MoveL BaseR_7,robotSpeed,fine,MoldGripper\WObj:=BaseMolds;
  ENDPROC
  PROC DropBlackL()
    MoveJ LeftHome,robotSpeed,z100,MoldGripper\WObj:=LeftMoldStore;
    MoveJ BlackL_6,robotSpeed,z100,MoldGripper\WObj:=LeftMoldStore;
    MoveL BlackL_5,robotSpeed,fine,MoldGripper\WObj:=LeftMoldStore;
    MoveL BlackL_4,robotSpeed,fine,MoldGripper\WObj:=LeftMoldStore;
    MoveL BlackL_3,robotSpeed,fine,MoldGripper\WObj:=LeftMoldStore;
    MoveL BlackL_2,robotSpeed,fine,MoldGripper\WObj:=LeftMoldStore;
    MoveJ BlackL_1,robotSpeed,z100,MoldGripper\WObj:=LeftMoldStore;
  ENDPROC
  PROC DropBlackR()
    MoveJ RightHome,robotSpeed,z100,MoldGripper\WObj:=RightMoldStore;
    MoveJ BlackR_6,robotSpeed,z100,MoldGripper\WObj:=RightMoldStore;
    MoveL BlackR_5,robotSpeed,fine,MoldGripper\WObj:=RightMoldStore;
    MoveL BlackR_4,robotSpeed,fine,MoldGripper\WObj:=RightMoldStore;
    MoveL BlackR_3,robotSpeed,fine,MoldGripper\WObj:=RightMoldStore;
    MoveL BlackR_2,robotSpeed,fine,MoldGripper\WObj:=RightMoldStore;
    MoveJ BlackR_1,robotSpeed,z100,MoldGripper\WObj:=RightMoldStore;
  ENDPROC
  PROC DropRedL()
    MoveJ LeftHome,robotSpeed,z100,MoldGripper\WObj:=LeftMoldStore;
    MoveJ RedL_6,robotSpeed,z100,MoldGripper\WObj:=LeftMoldStore;
    MoveL RedL_5,robotSpeed,fine,MoldGripper\WObj:=LeftMoldStore;
    MoveL RedL_4,robotSpeed,fine,MoldGripper\WObj:=LeftMoldStore;
    MoveL RedL_3,robotSpeed,fine,MoldGripper\WObj:=LeftMoldStore;
    MoveL RedL_2,robotSpeed,fine,MoldGripper\WObj:=LeftMoldStore;
    MoveJ RedL_1,robotSpeed,z100,MoldGripper\WObj:=LeftMoldStore;
  ENDPROC
  PROC DropRedR()
    MoveJ RightHome,v7000,z100,MoldGripper\WObj:=RightMoldStore;
    MoveJ RedR_6,robotSpeed,z100,MoldGripper\WObj:=RightMoldStore;
    MoveL RedR_5,robotSpeed,fine,MoldGripper\WObj:=RightMoldStore;
    MoveL RedR_4,robotSpeed,fine,MoldGripper\WObj:=RightMoldStore;
    MoveL RedR_3,robotSpeed,fine,MoldGripper\WObj:=RightMoldStore;
    MoveL RedR_2,robotSpeed,fine,MoldGripper\WObj:=RightMoldStore;
    MoveJ RedR_1,robotSpeed,z100,MoldGripper\WObj:=RightMoldStore;
  ENDPROC
  PROC DropBlueL()
    MoveJ LeftHome,robotSpeed,z100,MoldGripper\WObj:=LeftMoldStore;
    MoveJ BlueL_6,robotSpeed,z100,MoldGripper\WObj:=LeftMoldStore;
    MoveL BlueL_5,robotSpeed,fine,MoldGripper\WObj:=LeftMoldStore;
    MoveL BlueL_4,robotSpeed,fine,MoldGripper\WObj:=LeftMoldStore;
    MoveL BlueL_3,robotSpeed,fine,MoldGripper\WObj:=LeftMoldStore;
    MoveL BlueL_2,robotSpeed,fine,MoldGripper\WObj:=LeftMoldStore;
    MoveJ BlueL_1,robotSpeed,z100,MoldGripper\WObj:=LeftMoldStore;
  ENDPROC
  PROC DropBlueR()
    MoveJ RightHome,robotSpeed,z100,MoldGripper\WObj:=RightMoldStore;
    MoveJ BlueR_6,robotSpeed,z100,MoldGripper\WObj:=RightMoldStore;
    MoveL BlueR_5,robotSpeed,fine,MoldGripper\WObj:=RightMoldStore;
    MoveL BlueR_4,robotSpeed,fine,MoldGripper\WObj:=RightMoldStore;
    MoveL BlueR_3,robotSpeed,fine,MoldGripper\WObj:=RightMoldStore;
    MoveL BlueR_2,robotSpeed,fine,MoldGripper\WObj:=RightMoldStore;
    MoveJ BlueR_1,robotSpeed,z100,MoldGripper\WObj:=RightMoldStore;
  ENDPROC
  PROC velocity()
  ENDPROC
  PROC wait()
    WaitTime 16.5;
  ENDPROC
  PROC main()
    velocity;
    GoRest;
    GoHome;
    SetUpBlack_1;
    wait;
    TareDownBlack;
    SetUpRed;
    wait;
    TareDownRed;
    SetUpBlue;
    wait;
    TareDownBlue;
    SetUpBlack_2;
    GoHome;
  ENDPROC
  PROC SetUpRed()
    TakeRedR;
    DropOnBaseR;
    GoHome;
    TakeRedL;
    DropOnBaseL;
    GoHome;
  ENDPROC
  PROC SetUpBlue()
    TakeBlueR;
    DropOnBaseR;
    GoHome;
    TakeBlueL;
    DropOnBaseL;
    GoHome;
  ENDPROC
  PROC TareDownBlack()
    TakeFromBaseL;
    DropBlackL;
    GoHome;
    TakeFromBaseR;
    DropBlackR;
  ENDPROC
  PROC TareDownRed()
    TakeFromBaseL;
    DropRedL;
    GoHome;
    TakeFromBaseR;
    DropRedR;
  ENDPROC
  PROC TareDownBlue()
    TakeFromBaseL;
    DropBlueL;
    GoHome;
    TakeFromBaseR;
    DropBlueR;
  ENDPROC
  PROC SetUpBlack_1()
    TakeBlackL;
    DropOnBaseL;
    GoHome;
    TakeBlackR;
    DropOnBaseR;
    GoHome;
  ENDPROC
  PROC SetUpBlack_2()
    TakeBlackR;
    DropOnBaseR;
    GoHome;
    TakeBlackL;
    DropOnBaseL;
    GoHome;
  ENDPROC
ENDMODULE

! task T_ROB1
MODULE CalibData
  PERS tooldata MoldGripper:=[TRUE,[[-10.5,0,100],[1,0,0,0]],[1.873,[-1.681,0,-0.205],[1,0,0,0],0.002877912,0.002365912,0.002366511]];
  TASK PERS wobjdata BaseMolds:=[FALSE,TRUE,"",[[1700,200,1200],[0.5,-0.5,0.5,0.5]],[[0,0,0],[1,0,0,0]]];
  TASK PERS wobjdata LeftMoldStore:=[FALSE,TRUE,"",[[250,1550,1500],[0.5,-0.5,0.5,0.5]],[[0,0,0],[1,0,0,0]]];
  TASK PERS wobjdata RightMoldStore:=[FALSE,TRUE,"",[[-250,-1550,1500],[0.5,0.5,0.5,-0.5]],[[0,0,0],[1,0,0,0]]];
  CONST robtarget Home:=[[-175,1200,-200],[0.707106781,0.707106781,0,0],[0,0,0,0],[9E+09,9E+09,9E+09,9E+09,9E+09,9E+09]];
  CONST robtarget LeftHome:=[[175.014,250,-865],[1,0,0,0],[1,0,-1,0],[9E+09,9E+09,9E+09,9E+09,9E+09,9E+09]];
  CONST robtarget BlackL_1:=[[215.014,250,-110],[1,0,0,0],[1,-1,0,1],[9E+09,9E+09,9E+09,9E+09,9E+09,9E+09]];
  CONST robtarget BlackL_2:=[[215.014,250,-10],[1,0,0,0],[1,-1,0,1],[9E+09,9E+09,9E+09,9E+09,9E+09,9E+09]];
  CONST robtarget BlackL_3:=[[215.014,250,85],[1,0,0,0],[1,-1,0,1],[9E+09,9E+09,9E+09,9E+09,9E+09,9E+09]];
  CONST robtarget BlackL_4:=[[195.014,250,85],[1,0,0,0],[1,-1,0,1],[9E+09,9E+09,9E+09,9E+09,9E+09,9E+09]];
  CONST robtarget BlackL_5:=[[175.014,250,85],[1,0,0,0],[1,-1,0,1],[9E+09,9E+09,9E+09,9E+09,9E+09,9E+09]];
  CONST robtarget BlackL_6:=[[175.014,250,-315],[1,0,0,0],[1,-1,0,1],[9E+09,9E+09,9E+09,9E+09,9E+09,9E+09]];
  CONST robtarget BaseL_7:=[[-324.986,1250,-15],[1,0,0,0],[-1,1,-1,0],[9E+09,9E+09,9E+09,9E+09,9E+09,9E+09]];
  CONST robtarget BaseL_6:=[[-324.986,250,-15],[1,0,0,0],[-1,1,-1,0],[9E+09,9E+09,9E+09,9E+09,9E+09,9E+09]];
  CONST robtarget BaseL_5:=[[-324.986,250,85],[1,0,0,0],[0,0,-1,0],[9E+09,9E+09,9E+09,9E+09,9E+09,9E+09]];
  CONST robtarget BaseL_4:=[[-224.986,250,85],[1,0,0,0],[0,1,-2,0],[9E+09,9E+09,9E+09,9E+09,9E+09,9E+09]];
  CONST robtarget BaseL_3:=[[-204.986,250,85],[1,0,0,0],[0,1,-2,0],[9E+09,9E+09,9E+09,9E+09,9E+09,9E+09]];
  CONST robtarget BaseL_2:=[[-184.986,250,85],[1,0,0,0],[0,1,-2,0],[9E+09,9E+09,9E+09,9E+09,9E+09,9E+09]];
  CONST robtarget BaseL_1:=[[-184.986,250,-10],[1,0,0,0],[-1,0,-2,0],[9E+09,9E+09,9E+09,9E+09,9E+09,9E+09]];
  CONST robtarget BaseR_7:=[[-324.986,1250,-385],[0,1,0,0],[0,-2,0,0],[9E+09,9E+09,9E+09,9E+09,9E+09,9E+09]];
  CONST robtarget BaseR_6:=[[-324.986,250,-385],[0,1,0,0],[0,-2,0,0],[9E+09,9E+09,9E+09,9E+09,9E+09,9E+09]];
  CONST robtarget BaseR_5:=[[-324.986,250,-485],[0,1,0,0],[-1,-1,0,0],[9E+09,9E+09,9E+09,9E+09,9E+09,9E+09]];
  CONST robtarget BaseR_4:=[[-224.986,250,-485],[0,1,0,0],[-1,-2,1,0],[9E+09,9E+09,9E+09,9E+09,9E+09,9E+09]];
  CONST robtarget BaseR_3:=[[-204.986,250,-485],[0,1,0,0],[-1,-2,1,0],[9E+09,9E+09,9E+09,9E+09,9E+09,9E+09]];
  CONST robtarget BaseR_2:=[[-184.986,250,-485],[0,1,0,0],[-1,-2,1,0],[9E+09,9E+09,9E+09,9E+09,9E+09,9E+09]];
  CONST robtarget BaseR_1:=[[-184.986,250,-390],[0,1,0,0],[0,-1,1,0],[9E+09,9E+09,9E+09,9E+09,9E+09,9E+09]];
  CONST robtarget RightHome:=[[175.014,250,-765],[1,0,0,0],[-1,1,-2,1],[9E+09,9E+09,9E+09,9E+09,9E+09,9E+09]];
  CONST robtarget BlackR_1:=[[215.014,250,-110],[1,0,0,0],[-1,0,-1,1],[9E+09,9E+09,9E+09,9E+09,9E+09,9E+09]];
  CONST robtarget BlackR_2:=[[215.014,250,-10],[1,0,0,0],[-1,-1,0,1],[9E+09,9E+09,9E+09,9E+09,9E+09,9E+09]];
  CONST robtarget BlackR_3:=[[215.014,250,85],[1,0,0,0],[-1,-1,0,1],[9E+09,9E+09,9E+09,9E+09,9E+09,9E+09]];
  CONST robtarget BlackR_4:=[[195.014,250,85],[1,0,0,0],[-1,-1,0,1],[9E+09,9E+09,9E+09,9E+09,9E+09,9E+09]];
  CONST robtarget BlackR_5:=[[175.014,250,85],[1,0,0,0],[-1,-1,0,1],[9E+09,9E+09,9E+09,9E+09,9E+09,9E+09]];
  CONST robtarget BlackR_6:=[[175.014,250,-315],[1,0,0,0],[-1,-1,0,1],[9E+09,9E+09,9E+09,9E+09,9E+09,9E+09]];
  CONST robtarget RedL_1:=[[715.014,250,-110],[1,0,0,0],[1,-1,0,1],[9E+09,9E+09,9E+09,9E+09,9E+09,9E+09]];
  CONST robtarget RedL_2:=[[715.014,250,-10],[1,0,0,0],[1,-1,0,1],[9E+09,9E+09,9E+09,9E+09,9E+09,9E+09]];
  CONST robtarget RedL_3:=[[715.014,250,85],[1,0,0,0],[1,-1,0,1],[9E+09,9E+09,9E+09,9E+09,9E+09,9E+09]];
  CONST robtarget RedL_4:=[[695.014,250,85],[1,0,0,0],[1,-1,0,1],[9E+09,9E+09,9E+09,9E+09,9E+09,9E+09]];
  CONST robtarget RedL_5:=[[675.014,250,85],[1,0,0,0],[1,-1,0,1],[9E+09,9E+09,9E+09,9E+09,9E+09,9E+09]];
  CONST robtarget RedL_6:=[[675.014,250,-315],[1,0,0,0],[1,-1,0,1],[9E+09,9E+09,9E+09,9E+09,9E+09,9E+09]];
  CONST robtarget RedR_1:=[[715.014,250,-110],[1,0,0,0],[-1,0,-1,1],[9E+09,9E+09,9E+09,9E+09,9E+09,9E+09]];
  CONST robtarget RedR_2:=[[715.014,250,-10],[1,0,0,0],[-1,-1,0,1],[9E+09,9E+09,9E+09,9E+09,9E+09,9E+09]];
  CONST robtarget RedR_3:=[[715.014,250,85],[1,0,0,0],[-1,-1,0,1],[9E+09,9E+09,9E+09,9E+09,9E+09,9E+09]];
  CONST robtarget RedR_4:=[[695.014,250,85],[1,0,0,0],[-1,-1,0,1],[9E+09,9E+09,9E+09,9E+09,9E+09,9E+09]];
  CONST robtarget RedR_5:=[[675.014,250,85],[1,0,0,0],[-1,0,-1,1],[9E+09,9E+09,9E+09,9E+09,9E+09,9E+09]];
  CONST robtarget RedR_6:=[[675.014,250,-315],[1,0,0,0],[-1,0,-1,1],[9E+09,9E+09,9E+09,9E+09,9E+09,9E+09]];
  CONST robtarget BlueL_1:=[[1215.014,250,-110],[1,0,0,0],[1,0,0,1],[9E+09,9E+09,9E+09,9E+09,9E+09,9E+09]];
  CONST robtarget BlueL_2:=[[1215.014,250,-10],[1,0,0,0],[1,0,0,1],[9E+09,9E+09,9E+09,9E+09,9E+09,9E+09]];
  CONST robtarget BlueL_3:=[[1215.014,250,85],[1,0,0,0],[1,0,0,1],[9E+09,9E+09,9E+09,9E+09,9E+09,9E+09]];
  CONST robtarget BlueL_4:=[[1195.014,250,85],[1,0,0,0],[1,0,0,1],[9E+09,9E+09,9E+09,9E+09,9E+09,9E+09]];
  CONST robtarget BlueL_5:=[[1175.014,250,85],[1,0,0,0],[1,0,0,1],[9E+09,9E+09,9E+09,9E+09,9E+09,9E+09]];
  CONST robtarget BlueL_6:=[[1175.014,250,-315],[1,0,0,0],[1,0,0,1],[9E+09,9E+09,9E+09,9E+09,9E+09,9E+09]];
  CONST robtarget BlueR_1:=[[1215.014,250,-110],[1,0,0,0],[-1,0,-1,1],[9E+09,9E+09,9E+09,9E+09,9E+09,9E+09]];
  CONST robtarget BlueR_2:=[[1215.014,250,-10],[1,0,0,0],[-1,0,0,1],[9E+09,9E+09,9E+09,9E+09,9E+09,9E+09]];
  CONST robtarget BlueR_3:=[[1215.014,250,85],[1,0,0,0],[-1,0,0,1],[9E+09,9E+09,9E+09,9E+09,9E+09,9E+09]];
  CONST robtarget BlueR_4:=[[1195.014,250,85],[1,0,0,0],[-1,0,0,1],[9E+09,9E+09,9E+09,9E+09,9E+09,9E+09]];
  CONST robtarget BlueR_5:=[[1175.014,250,85],[1,0,0,0],[-1,0,-1,1],[9E+09,9E+09,9E+09,9E+09,9E+09,9E+09]];
  CONST robtarget BlueR_6:=[[1175.014,250,-315],[1,0,0,0],[-1,0,0,1],[9E+09,9E+09,9E+09,9E+09,9E+09,9E+09]];
ENDMODULE

! task T_ROB1
MODULE Module1
  PROC TakeBlackLeft()
  ENDPROC
  PROC main()
    GoHome;
    CycleBlack;
    CycleRed;
    CycleBlue;
    GoHome;
  ENDPROC
  PROC GoHome()
  ENDPROC
  PROC LetBaseLeft()
  ENDPROC
  PROC LetBaseRight()
  ENDPROC
  PROC TakeBlackRight()
  ENDPROC
  PROC TakeRedLeft()
  ENDPROC
  PROC TakeRedRight()
  ENDPROC
  PROC TakeBlueLeft()
  ENDPROC
  PROC TakeBlueRight()
  ENDPROC
  PROC TakeBaseLeft()
  ENDPROC
  PROC TakeBaseRight()
  ENDPROC
  PROC LetBlackLeft()
    TakeBlackLeft;
    LetBaseLeft;
  ENDPROC
  PROC LetBlackRight()
    TakeBlackRight;
    LetBaseRight;
  ENDPROC
  PROC LetRedLeft()
    TakeRedLeft;
    LetBaseLeft;
  ENDPROC
  PROC LetRedRight()
    TakeRedRight;
    LetBaseRight;
  ENDPROC
  PROC LetBlueLeft()
    TakeBlueLeft;
    LetBaseLeft;
  ENDPROC
  PROC LetBlueRight()
    TakeBlueRight;
    LetBaseRight;
  ENDPROC
  PROC ReturnBlackLeft()
  ENDPROC
  PROC ReturnBlackRight()
  ENDPROC
  PROC ReturnRedLeft()
  ENDPROC
  PROC ReturnRedRight()
  ENDPROC
  PROC ReturnBlueLeft()
  ENDPROC
  PROC ReturnBlueRight()
  ENDPROC
  PROC BackBlackLeft()
    TakeBaseLeft;
    ReturnBlackLeft;
  ENDPROC
  PROC BackBlackRight()
    TakeBaseRight;
    ReturnBlackRight;
  ENDPROC
  PROC BackRedLeft()
    TakeBaseLeft;
    ReturnRedLeft;
  ENDPROC
  PROC BackRedRight()
    TakeBaseRight;
    ReturnRedRight;
  ENDPROC
  PROC BackBlueLeft()
    TakeBaseLeft;
    ReturnBlueLeft;
  ENDPROC
  PROC BackBlueRight()
    TakeBaseRight;
    ReturnBlueRight;
  ENDPROC
  PROC CycleBlack()
    LetBlackLeft;
    LetBlackRight;
    WaitTime 23;
    BackBlackLeft;
    BackBlackRight;
  ENDPROC
  PROC CycleRed()
    LetRedLeft;
    LetRedRight;
    WaitTime 23;
    BackRedLeft;
    BackRedRight;
  ENDPROC
  PROC CycleBlue()
    LetBlueLeft;
    LetBlueRight;
    WaitTime 23;
    BackBlueLeft;
    BackBlueRight;
  ENDPROC
ENDMODULE

